// TIA Portal V17 export
// export: Created 2025-08-05T09:36:02.210752Z, ExportSetting WithDefaults, DisplayName Totally Integrated Automation Portal, DisplayVersion V17, DisplayName TIA Portal Openness, DisplayVersion V17, DisplayName TIA Portal Version Control Interface, DisplayVersion V17, DisplayName SINAMICS Startdrive Advanced, DisplayVersion V17, DisplayName SINAMICS Startdrive G130, G150, S120, S150, SINAMICS MV, S210, DisplayVersion V17, DisplayName SINAMICS Startdrive G110M, G120, G120C, G120D, G120P, G115D, DisplayVersion V17, DisplayName STEP 7 Professional, DisplayVersion V17, DisplayName STEP 7 Safety, DisplayVersion V17, DisplayName WinCC Advanced, DisplayVersion V17
TYPE "LaserComm_LDD_Results"
// stored: IsFailsafeCompliant false
   STRUCT
      QA : DInt;   // Pass/Fail for the LDD Job (0= Incomplete, 1=Pass, 2= Fail, 3=No QA)
      Warning : DInt;   // Warning Code for the LDD Job (0= Incomplete, 1=Pass, 2= Fail, 3=No QA)
      Reasons : Struct   // Reason for Weld QA Failure
         KHD : DInt;   // Keyhole Depth Measurement
         FWS : DInt;   // Finished Weld Surface Measurement
         XSP : DInt;   // Cross Section Parameter Measurement
         SPO : DInt;   // Seam Position Measurement
         SLE : DInt;   // Seam Left Edge Measurement
         SRE : DInt;   // Seam Right Edge Measurement
         SLH : DInt;   // Seam Left Height Measurement
         SRH : DInt;   // Seam Right Height Measurement
         SHH : DInt;   // Seam Step Height Measurement
         SCP : DInt;   // Seam Centre Position Measurement
         SGP : DInt;   // Seam Gap Width Measurement
         SJP : DInt;   // Seam Joint Feature Position Measurement
         SJH : DInt;   // Seam Joint Feature Height Measurement
         WPH : DInt;   // Workpiece Height Measurement
         TLE : DInt;   // Transverse Profile Left Edge Position Measurement
         TRE : DInt;   // Transverse Profile Right Edge Position Measurement
         TBD : DInt;   // Weld Bead Centre Measurement
         TBW : DInt;   // Weld Bead Width Measurement
      END_STRUCT;
   END_STRUCT;
END_TYPE
